(* Logix 5000 project; controller PROCESS_OUTPUT Emulate 5570 rev 36.11; software revision 36.00 *)

TASK MainTask (continuous, watchdog 500 ms) : MainProgram

MODULES
   Local : Emulate 5570 (ICP 2, rev 36.11)
       : 1756-IB16 (ICP 3, rev 3.1, Input RPI 20 ms)
       : vendor 1 type 7 code 16 (ICP 4, rev 3.1, Output RPI 20 ms)
END_MODULES

VAR_GLOBAL   (* controller tags *)
   PROCESS_OUTPUT : ALIAS FOR Local:4:O.Data.0;   // Process Output
   SW_START : ALIAS FOR Local:3:I.Data.0;   // START Momentary N.O. Pushbutton
END_VAR

PROGRAM MainProgram   (* main routine MainRoutine *)
VAR
   A_MATERIAL_MULTIPLIER : REAL;   // Material A Multiplier
   B_MATERIAL_MULTIPLIER : REAL;   // Material B Multiplier
   C_MATERIAL_MULTIPLIER : REAL;   // Material C Multiplier
   D_MATERIAL_MULTIPLIER : REAL;   // Material D Multiplier
   HMI_A_MATERIAL_MULTIPLIER : ALIAS FOR A_MATERIAL_MULTIPLIER;
   HMI_ACC_PROCESS_TIME : ALIAS FOR PROCESS_TIME.ACC;
   HMI_B_MATERIAL_MULTIPLIER : ALIAS FOR B_MATERIAL_MULTIPLIER;
   HMI_C_MATERIAL_MULTIPLIER : ALIAS FOR C_MATERIAL_MULTIPLIER;
   HMI_D_MATERIAL_MULTIPLIER : ALIAS FOR D_MATERIAL_MULTIPLIER;
   HMI_NUM_SHEETS : ALIAS FOR NUM_SHEETS;
   HMI_PRE_PROCESS_TIME : ALIAS FOR PROCESS_TIME.PRE;
   HMI_TYPE_SHEETS : ALIAS FOR TYPE_SHEET;
   MATERIAL_MULTI_VALUE : REAL;   // Material Multplier Value
   NUM_SHEETS : INT;   // Value for Sheet Type
   PROCESS_TIME : TIMER;
   PROCESS_VALUE : REAL;   // Process Value
   TYPE_SHEET : INT;   // Value Number of Sheets
END_VAR

ROUTINE HMI_Routine   (* ladder *)
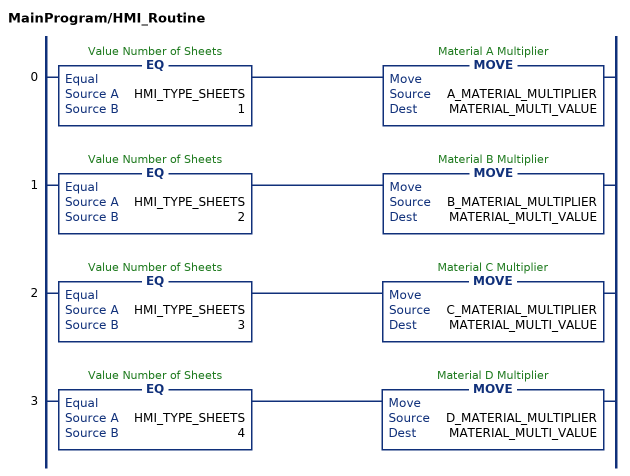
   0: EQ(HMI_TYPE_SHEETS,1)MOVE(A_MATERIAL_MULTIPLIER,MATERIAL_MULTI_VALUE);
   1: EQ(HMI_TYPE_SHEETS,2)MOVE(B_MATERIAL_MULTIPLIER,MATERIAL_MULTI_VALUE);
   2: EQ(HMI_TYPE_SHEETS,3)MOVE(C_MATERIAL_MULTIPLIER,MATERIAL_MULTI_VALUE);
   3: EQ(HMI_TYPE_SHEETS,4)MOVE(D_MATERIAL_MULTIPLIER,MATERIAL_MULTI_VALUE);
END_ROUTINE

ROUTINE MainRoutine   (* ladder *)
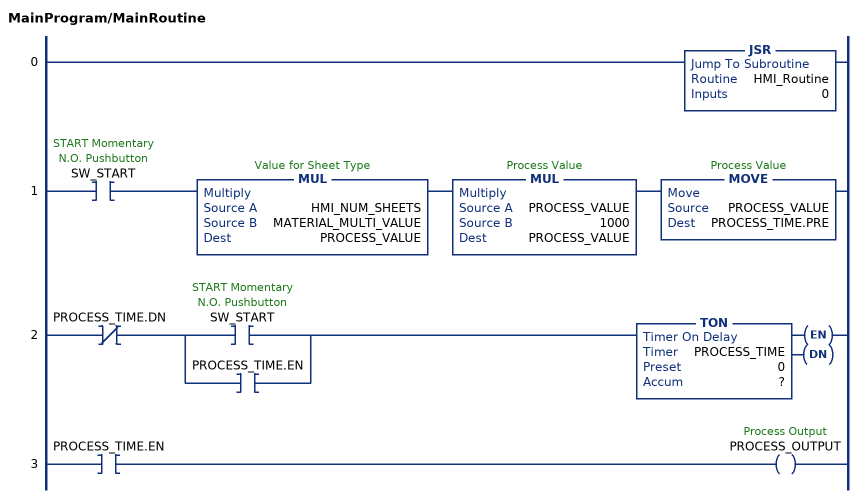
   0: JSR(HMI_Routine,0);
   1: XIC(SW_START)MUL(HMI_NUM_SHEETS,MATERIAL_MULTI_VALUE,PROCESS_VALUE)MUL(PROCESS_VALUE,1000,PROCESS_VALUE)MOVE(PROCESS_VALUE,PROCESS_TIME.PRE);
   2: XIO(PROCESS_TIME.DN)[XIC(SW_START) ,XIC(PROCESS_TIME.EN) ]TON(PROCESS_TIME,?,?);
   3: XIC(PROCESS_TIME.EN)OTE(PROCESS_OUTPUT);
END_ROUTINE
END_PROGRAM
